FUNCTION_BLOCK fbMultipleArmAgiCtrl
VAR_INPUT
	bEN: BOOL;
	bBasketCfm: BOOL;
	bEmergencyStop: BOOL;
	bStnProcessComplete: BOOL;
	bMultiArmAgiDownRS: BOOL;
	bMultiArmAgiMidRS: BOOL;
END_VAR
VAR_OUTPUT
	bMultiArmAgiInProcess: BOOL;
	bMultiArmAgiDown: BOOL;
	bMultiArmAgiUp: BOOL;

END_VAR
VAR

END_VAR

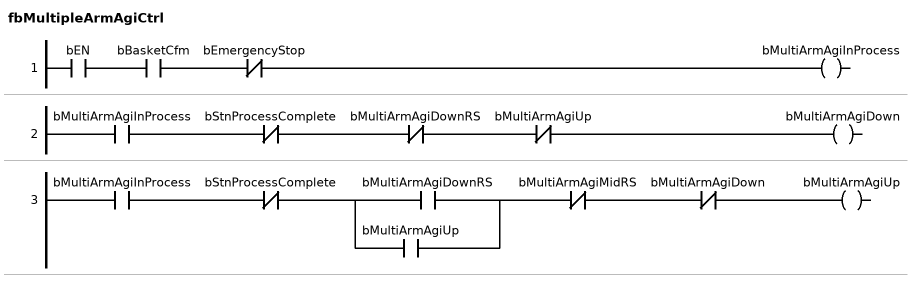
// NETWORK 1
bMultiArmAgiInProcess := bEN AND bBasketCfm AND NOT bEmergencyStop;

// NETWORK 2
bMultiArmAgiDown := bMultiArmAgiInProcess AND NOT bStnProcessComplete AND NOT bMultiArmAgiDownRS AND NOT bMultiArmAgiUp;

// NETWORK 3
bMultiArmAgiUp := (bMultiArmAgiInProcess AND NOT bStnProcessComplete AND (bMultiArmAgiDownRS OR bMultiArmAgiUp)) AND NOT bMultiArmAgiMidRS AND NOT bMultiArmAgiDown;

END_FUNCTION_BLOCK

(* stored: Version 1.1.0.1, ProductVersion 3.1.4024.12
   POU fbMultipleArmAgiCtrl: Id {2c22ed7f-59a7-492e-a2e6-cb6df421e1e8}, SpecialFunc None *)
